(* IEC 61131-3 sources: ATCMcontrol_Engineering/src/TargetBase/Libs/MBRTU, 20 files *)

(* ---- MB_data.st ---- *)
(*[[
    UserHelpURL= "ATCMfile:MB_data.HTML",
]]*)
FUNCTION MB_data : UINT
VAR_OUTPUT
	data : ARRAY[0..257] OF UINT; (*[return value]*)
END_VAR
INLINE {STDLIB(MB_data)}
END_FUNCTION

(* ---- MB_f01.st ---- *)
(*[[
    UserHelpURL= "ATCMfile:MB_f01.HTML",
    UserText1= "fn_01_read_coil_status",
]]*)
FUNCTION MB_f01 : UINT
VAR_INPUT
	slave      : UINT; (*[slave number]*)
    start_addr : UINT; (*[start address]*)
    count      : UINT; (*[counter]*)
END_VAR
INLINE {STDLIB(MB_f01)}
END_FUNCTION

(* ---- MB_f02.st ---- *)
(*[[
    UserHelpURL= "ATCMfile:MB_f02.HTML",
    UserText1= "fn_02_read_input_status",
]]*)
FUNCTION MB_f02 : UINT
VAR_INPUT
	slave      : UINT; (*[slave number]*)
    start_addr : UINT; (*[start address]*)
    count      : UINT; (*[counter]*)
END_VAR
INLINE {STDLIB(MB_f02)}
END_FUNCTION

(* ---- MB_f03.st ---- *)
(*[[
    UserHelpURL= "ATCMfile:MB_f03.HTML",
    UserText1= "fn_03_read_holding_register",
]]*)
FUNCTION MB_f03 : UINT
VAR_INPUT
	slave      : UINT; (*[slave number]*)
    start_addr : UINT; (*[start address]*)
    count      : UINT; (*[counter]*)
    byteorder  : UINT; (*[byte order]*)
END_VAR
INLINE {STDLIB(MB_f03)}
END_FUNCTION

(* ---- MB_f04.st ---- *)
(*[[
    UserHelpURL= "ATCMfile:MB_f04.HTML",
    UserText1= "fn_04_read_input_registers",
]]*)
FUNCTION MB_f04 : UINT
VAR_INPUT
	slave      : UINT; (*[slave number]*)
    start_addr : UINT; (*[start address]*)
    count      : UINT; (*[counter]*)
    byteorder  : UINT; (*[byte order]*)
END_VAR
INLINE {STDLIB(MB_f04)}
END_FUNCTION

(* ---- MB_f05.st ---- *)
(*[[
    UserHelpURL= "ATCMfile:MB_f05.HTML",
    UserText1= "fn_05_force_single_coil",
]]*)
FUNCTION MB_f05 : UINT
VAR_INPUT
	slave      : UINT; (*[slave number]*)
    coil_addr  : UINT; (*[coil address]*)
    coil_state : UINT; (*[coil state]*)
END_VAR
INLINE {STDLIB(MB_f05)}
END_FUNCTION

(* ---- MB_f06.st ---- *)
(*[[
    UserText1= "fn_06_preset_single_register",
    UserHelpURL= "ATCMfile:MB_f06.HTML",
]]*)
FUNCTION MB_f06 : UINT
VAR_INPUT
	slave      : UINT; (*[slave number]*)
    reg_addr   : UINT; (*[register address]*)
	value      : UINT; (*[value to set]*)
END_VAR
INLINE {STDLIB(MB_f06)}
END_FUNCTION

(* ---- MB_f07.st ---- *)
(*[[
    UserHelpURL= "ATCMfile:MB_f07.HTML",
    UserText1= "fn_07_read_exception_status",
]]*)
(*
Return bits:
[0] = Number of the exception status coils (8);
[1] = exception status  coil1  value (ON/OFF)
[2] = exception status  coil2  value (ON/OFF) ...
*)
FUNCTION MB_f07 : UINT
VAR_INPUT
	slave      : UINT; (*[slave number]*)
END_VAR
INLINE {STDLIB(MB_f07)}
END_FUNCTION

(* ---- MB_f08.st ---- *)
(*[[
    UserHelpURL= "ATCMfile:MB_f08.HTML",
    UserText1= "fn_08_diagnostics",
]]*)
FUNCTION MB_f08 : UINT
VAR_INPUT
	slave      : UINT; (*[slave number]*)
	subfunction: UINT; (*[sub-function pointer to test]*)
END_VAR
INLINE {STDLIB(MB_f08)}
END_FUNCTION

(* ---- MB_f0b.st ---- *)
(*[[
    UserHelpURL= "ATCMfile:MB_f0b.HTML",
    UserText1= "fn_0b_read_event_counter",
]]*)
(*
Return bits:
[0] = status word
[1] = event count
*)
FUNCTION MB_f0b : UINT
VAR_INPUT
	slave      : UINT; (*[slave number]*)
END_VAR
INLINE {STDLIB(MB_f0b)}
END_FUNCTION

(* ---- MB_f0c.st ---- *)
(*[[
    UserHelpURL= "ATCMfile:MB_f0c.HTML",
    UserText1= "fn_0c_read_event_log",
]]*)
(*
Return bits:
[0] = Number of event (0-64)
[1] = Status Word
[2] = Event Count
[3] = Message Count
[4] = Event 0 byte
[5] = Event 1 byte ....
*)
FUNCTION MB_f0c : UINT
VAR_INPUT
	slave      : UINT; (*[slave number]*)
END_VAR
INLINE {STDLIB(MB_f0c)}
END_FUNCTION

(* ---- MB_f0f.st ---- *)
(*[[
    UserHelpURL= "ATCMfile:MB_f0f.HTML",
    UserText1= "fn_0f_force_multiple_coil",
]]*)
FUNCTION MB_f0f : UINT
VAR_INPUT
	slave      : UINT; (*[slave number]*)
    coil_addr  : UINT; (*[coil address]*)
    coil_count : UINT; (*[coil counter]*)
    values : ARRAY[0..257] of UINT; (*[coils values to force]*)
END_VAR
INLINE {STDLIB(MB_f0f)}
END_FUNCTION

(* ---- MB_f10.st ---- *)
(*[[
    UserText1= "fn_10_preset_multiple_registers",
    UserHelpURL= "ATCMfile:MB_f10.HTML",
]]*)
FUNCTION MB_f10 : UINT
VAR_INPUT
	slave      : UINT; (*[slave number]*)
    start_addr : UINT; (*[start address]*)
    count      : UINT; (*[counter]*)
    value : ARRAY[0..257] of UINT; (*[registers value to set]*)
END_VAR
INLINE {STDLIB(MB_f10)}
END_FUNCTION

(* ---- MB_f11.st ---- *)
(*[[
    UserText1= "fn_11_report_slave_id",
    UserHelpURL= "ATCMfile:MB_f11.HTML",
]]*)
(*
Return bits:
[0] = # of the received byte, each of them is stored in the following array location
      in the same arrangement they are received
[i] = data byte
*)
FUNCTION MB_f11 : UINT
VAR_INPUT
	slave      : UINT; (*[slave number]*)
END_VAR
INLINE {STDLIB(MB_f11)}
END_FUNCTION

(* ---- MB_f14.st ---- *)
(*[[
    UserText1= "fn_14_read_general_reference",
    UserHelpURL= "ATCMfile:MB_f14.HTML",
]]*)
 (*
Return bits:
 [0] = the total number of valid entries in the following array location
 [1] = # of data N for group reference 1
 [2] = data0 for group reference 1
 [3] = data1 for group reference 1
 .....
 [K] = dataN for group reference 1
 [K+1] = # of data M for group reference 2
 [K+2] = data0 for group reference 2
 .....
 [H] = dataM for group reference 2
*)
FUNCTION MB_f14 : UINT
VAR_INPUT
	slave      : UINT; (*[slave number]*)
(*
[0] = number of group of refrence to be read (from 1 ...to N)
[1] = extended Memory file number for group 1
[2] = starting register address for group 1
[3] = quantity of registers to be read for group 1
[4] = extended Memory file number for group 2
[5] = starting register address for group 2
[6] = quantity of registers to be read for group 2
...
*)
    query : ARRAY[0..257] of UINT; (*[query]*)
END_VAR
INLINE {STDLIB(MB_f14)}
END_FUNCTION

(* ---- MB_f15.st ---- *)
(*[[
    UserText1= "fn_15_write_general_reference",
    UserHelpURL= "ATCMfile:MB_f15.HTML",
]]*)
FUNCTION MB_f15 : UINT
VAR_INPUT
	slave      : UINT; (*[slave number]*)
    count      : UINT; (*[counter]*)
(*
[0] = 0x06 the reference type fixed to 0x0006
[1] = Extended Memory file number (1 to 10, hex 0001 to 000A);
[2] = starting register address within the file
[3] = quantity of registers to be written
[4] =  data to be written
[5] =  data to be written
[6] =  data to be written
[7] =  data to be written
....
[n] = 0x06 the reference type fixed to 0x0006
[n+1] = Extended Memory file number (1 to 10, hex 0001 to 000A);
[n+2] = starting register address within the file
[n+3] = quantity of registers to be written
[n+4] =  data to be written
[n+5] =  data to be written
[n+6] =  data to be written
[n+7] =  data to be written
*)
    data : ARRAY[0..257] of UINT; (*[data to write]*)
END_VAR
INLINE {STDLIB(MB_f15)}
END_FUNCTION

(* ---- MB_f16.st ---- *)
(*[[
    UserText1= "fn_16_mask_write_registers",
    UserHelpURL= "ATCMfile:MB_f16.HTML",
]]*)
FUNCTION MB_f16 : UINT
VAR_INPUT
	slave      : UINT; (*[slave number]*)
    start_addr : UINT; (*[start address]*)
(*
[0] = And Mask
[1] = Or Mask
*)
    data : ARRAY[0..2] of UINT; (*[0 = And Mask; 1 = Or Mask]*)
END_VAR
INLINE {STDLIB(MB_f16)}
END_FUNCTION

(* ---- MB_f17.st ---- *)
(*[[
    UserText1= "fn_17_read_write_registers",
    UserHelpURL= "ATCMfile:MB_f17.HTML",
]]*)
FUNCTION MB_f17 : UINT
(*
Return bits:

*)
VAR_INPUT
	slave      : UINT; (*[slave number]*)
    start_addr : UINT; (*[start address]*)
    count      : UINT; (*[counter]*)
    reg_addr   : UINT; (*[register address]*)
    byteorder  : BYTE; (*[byte order]*)
    data : ARRAY[0..257] of UINT; (*[value to write]*)
END_VAR
INLINE {STDLIB(MB_f17)}
END_FUNCTION

(* ---- MB_f18.st ---- *)
(*[[
    UserText1= "fn_18_read_fifo_queue",
    UserHelpURL= "ATCMfile:MB_f18.HTML",
]]*)
(*
Return bits:
all
*)
FUNCTION MB_f18 : UINT
VAR_INPUT
	slave      : UINT; (*[slave number]*)
    start_addr : UINT; (*[start address]*)
END_VAR
INLINE {STDLIB(MB_f18)}
END_FUNCTION

(* ---- MB_get_status.st ---- *)
(*[[
    UserHelpURL= "ATCMfile:MB_get_status.HTML",
]]*)
FUNCTION MB_get_status : UINT
VAR_OUTPUT
    data : ARRAY[0..2] of UINT; (*[return value]*)
END_VAR
INLINE {STDLIB(MB_get_status)}
END_FUNCTION
